FUNCTION_BLOCK FB_IoLinkPatlite EXTENDS FB_IolStdVarSlave IMPLEMENTS I_Patlite
VAR
	bBuzzerON			AT %Q*	:BOOL;					//ブザー出力
	bRedTier			AT %Q*	:BOOL;					//RedLED出力
	bYellowTier			AT %Q*	:BOOL;					//YellowLED出力
	bGreenTier			AT %Q*	:BOOL;					//GreenLED出力
	bBlueTier			AT %Q*	:BOOL;					//BlueLED出力
	bWhiteTier			AT %Q*	:BOOL;					//WhiteLED出力
	
	bBuzzerFlag					:BOOL;					//ブザー停止記憶
	
	fbStartupBuzzerREdge		:R_TRIG;
	fbStartupBuzzerFEdge		:F_TRIG;
	
	hr							:HRESULT;
	fbhrTon						:ton:=(PT:=T#1S);
	
	usiBuzzerPattern			:USINT;
	usiReadBuzzerPattern		:USINT;

	iStep						:INT;
	ePrevMachineState			:E_MachineState;
	
END_VAR

(*
パトライトのLB6-20ILWCBW用FB

初期化の際にIO-LinkマスターのAoE Net IDと接続先ポートナンバーとデバイス名を設定して下さい。
この三項目を設定しないとFB_IolStdVarSlaveのメソッドが使えません。

*)

PROPERTY bBuzzerStop : BOOL
SET
//---スイッチが押されたらブザー停止---
	IF bBuzzerStop=TRUE THEN
		bBuzzerON:=FALSE;
		bBuzzerFlag:=TRUE;
	END_IF
END_SET
END_PROPERTY

PROPERTY bStartupBuzzer : BOOL
SET
fbStartupBuzzerREdge(CLK:=bStartupBuzzer);
fbStartupBuzzerFEdge(CLK:=bStartupBuzzer);

IF fbStartupBuzzerREdge.Q=TRUE THEN
	iStep:=1;
	usiBuzzerPattern	:=8;		//スイープ音（ヒューン）500ms ON / 500ms OFF
	bBuzzerON:=TRUE;
	bBuzzerFlag:=FALSE;
ELSIF fbStartupBuzzerFEdge.Q=TRUE THEN
	iStep:=1;
	usiBuzzerPattern	:=3;		//高低音（ピポピポ）
	bBuzzerON:=FALSE;
END_IF


//---パラメーターを書き換え---

(*
fbhrTon(IN:= hr=16#203);
IF fbhrTon.Q THEN
	iStep:=iStep +1;
END_IF
*)

CASE iStep OF
	0:
		(*NA*)
	1:
		hr:=SUPER^.Write_UINT8(	nIndex		:=16#07EE,	//Buzzer Pattern
								nSubindex	:=16#00,
								nData		:=usiBuzzerPattern);					

		IF NOT F_IolIsBusy(hr) THEN
				iStep:=2;
		 END_IF
	
	2:
		hr:=SUPER^.Read_UINT8(	nIndex		:=16#07EE,	//Buzzer Pattern
								nSubindex	:=16#00,
								nData		:=usiReadBuzzerPattern);
								
		IF NOT F_IolIsBusy(hr) THEN
			iStep:=3;
		END_IF
	
	3:
		IF usiReadBuzzerPattern<>usiBuzzerPattern THEN
			iStep:=1;
		ELSE
			iStep:=0;
		END_IF

END_CASE
END_SET
END_PROPERTY

PROPERTY eMachineState : E_MachineState
SET
//---マシーンステートごとにパトライトを制御---

	IF ePrevMachineState<>eMachineState THEN
		bBuzzerON:=FALSE;
		bBuzzerFlag:=FALSE;
		ePrevMachineState:=eMachineState;
	END_IF

	CASE eMachineState OF
		
		E_MachineState.Critical:
			IF bBuzzerFlag=FALSE THEN
				bBuzzerON:=TRUE;
			END_IF
		
			bRedTier			:=TRUE;
			bYellowTier			:=FALSE;
			bGreenTier			:=FALSE;
			bBlueTier			:=TRUE;
			bWhiteTier			:=FALSE;
		
		E_MachineState.Error:
			IF bBuzzerFlag=FALSE THEN
				bBuzzerON:=TRUE;
			END_IF
		
			bRedTier			:=TRUE;
			bYellowTier			:=FALSE;
			bGreenTier			:=FALSE;
			bBlueTier			:=FALSE;
			bWhiteTier			:=FALSE;

		E_MachineState.Warning:
			IF bBuzzerFlag=FALSE THEN
				bBuzzerON:=TRUE;
			END_IF
		
			bRedTier			:=FALSE;
			bYellowTier			:=TRUE;
			bGreenTier			:=FALSE;
			bBlueTier			:=FALSE;
			bWhiteTier			:=FALSE;

			
		E_MachineState.Stay:
			bRedTier			:=FALSE;
			bYellowTier			:=FALSE;
			bGreenTier			:=FALSE;
			bBlueTier			:=FALSE;
			bWhiteTier			:=TRUE;
		
		E_MachineState.Stop:
			bRedTier			:=FALSE;
			bYellowTier			:=FALSE;
			bGreenTier			:=TRUE;
			bBlueTier			:=FALSE;
			bWhiteTier			:=TRUE;
	
		E_MachineState.Moving:
			bRedTier			:=FALSE;
			bYellowTier			:=FALSE;
			bGreenTier			:=TRUE;
			bBlueTier			:=FALSE;
			bWhiteTier			:=FALSE;

	END_CASE;
END_SET
END_PROPERTY

//FB_Init は常に暗黙的に使用可能で、主に初期化に使用されます。
//戻り値は評価されません。特定の結果を得るために、メソッドを明示的に宣言し、
//そのメソッドに標準の初期化コードをもったコードを追加することができます。戻り値を評価できます。
METHOD FB_Init: BOOL
VAR_INPUT
    bInitRetains: BOOL; // TRUE: 保持変数は初期化されます (ウォーム リセット、あるいはコールド リセット)
    bInCopyCode: BOOL;  // TRUE: 後でコードをコピーする (オンライン変更) ために、インスタンスをコピーします。
	
	MasterAoeNetId	:T_AmsNetID;
	port			:E_IolPort;
	Name			:STRING(255);

END_VAR
SUPER^.MasterAoeNetId	:=MasterAoeNetId;
SUPER^.Port				:=port;
SUPER^.Name				:=Name;
END_METHOD

END_FUNCTION_BLOCK

(* stored: Version 1.1.0.1, ProductVersion 3.1.4026.13
   POU FB_IoLinkPatlite: Id {4e9b2e93-da1e-4356-8935-86acc05a1acf}, SpecialFunc None
   Property bBuzzerStop: Id {fba2f8e5-1b13-4c90-b931-e83614d5b6be}
   Set Set: Id {342385f4-e76c-4fe7-9b79-e4d8db2af8e1}
   Property bStartupBuzzer: Id {a03f1a37-4527-46a0-b6fa-c76e060636d0}
   Set Set: Id {7e1b0de0-7d42-4a70-9873-d93682e5d278}
   Property eMachineState: Id {b8041fad-c182-4001-b77a-fee831d6da20}
   Set Set: Id {fb29542b-6c65-4365-80f4-1f4495a514f0}
   Method FB_Init: Id {2606a8d6-f628-4022-8b12-3c6446bb2570} *)
